// TIA Portal V18 export
VAR_GLOBAL   // PLC tag table "17_AE1-SA2"
   "iAE1-SA2p" AT %I9.4 : Bool;   // 4
   "iAE1-SA2" AT %I9.5 : Bool;   // 4
   "iAE1-SA2a" AT %I17.4 : Bool;
   "oAE1-SA2p" AT %Q8.7 : Bool;
   "oAE1-SA2" AT %Q9.0 : Bool;
END_VAR
